     VAL_STRG(FORMAT := #CONVERT_FORMAT_TO_STRING,
              IN     := #date.MONTH,
              P      := #CONVERT_START_POSITION_MONTH,
              PREC   := #CONVERT_PRECISION,
              SIZE   := #CONVERT_SIZE_MONTH_DAY_HOUR_MINUTE_SECOND,
              OUT    => #tempString);     // DTL MONTH --> String --> #tempPosMonth

     VAL_STRG(FORMAT := #CONVERT_FORMAT_TO_STRING,
              IN     := #date.DAY,
              P      := #CONVERT_START_POSITION_DAY,
              PREC   := #CONVERT_PRECISION,
              SIZE   := #CONVERT_SIZE_MONTH_DAY_HOUR_MINUTE_SECOND,
              OUT    => #tempString);     // DTL DAY --> String --> #tempPosDay

     VAL_STRG(FORMAT := #CONVERT_FORMAT_TO_STRING,
              IN     := #date.HOUR,
              P      := #CONVERT_START_POSITION_HOUR,
              PREC   := #CONVERT_PRECISION,
              SIZE   := #CONVERT_SIZE_MONTH_DAY_HOUR_MINUTE_SECOND,
              OUT    => #tempString);     // DTL HOUR --> String --> #tempPosHour

     VAL_STRG(FORMAT := #CONVERT_FORMAT_TO_STRING,
              IN     := #date.MINUTE,
              P      := #CONVERT_START_POSITION_MINUTE,
              PREC   := #CONVERT_PRECISION,
              SIZE   := #CONVERT_SIZE_MONTH_DAY_HOUR_MINUTE_SECOND,
              OUT    => #tempString);     // DTL MINUTE --> String --> #tempPosMinute

     VAL_STRG(FORMAT := #CONVERT_FORMAT_TO_STRING,
              IN     := #date.SECOND,
              P      := #CONVERT_START_POSITION_SECOND,
              PREC   := #CONVERT_PRECISION,
              SIZE   := #CONVERT_SIZE_MONTH_DAY_HOUR_MINUTE_SECOND,
              OUT    => #tempString);     // DTL SECOND --> String --> #tempPosSecond

     VAL_STRG(FORMAT := #CONVERT_FORMAT_TO_STRING,
              IN     := #date.NANOSECOND,
              P      := #CONVERT_START_POSITION_NANOSECOND,
              PREC   := #CONVERT_PRECISION,
              SIZE   := #CONVERT_SIZE_NANOSECOND,
              OUT    => #tempString);     // DTL NANOSECOND --> String --> #tempPosNanosecond

     // Place separators at the right position in the string
     IF #separator = '' THEN
       #tempString[#SEPARATOR_POSITION_YEAR_MONTH] := #SEPARATOR_DATE;
       #tempString[#SEPARATOR_POSITION_MONTH_DAY] := #SEPARATOR_DATE;
     ELSE
       #tempString[#SEPARATOR_POSITION_YEAR_MONTH] := #separator;
       #tempString[#SEPARATOR_POSITION_MONTH_DAY] := #separator;
     END_IF;
     #tempString[#SEPARATOR_POSITION_HOUR_MINUTE] := #SEPARATOR_TIME;
     #tempString[#SEPARATOR_POSITION_MINUTE_SECOND] := #SEPARATOR_TIME;
     #tempString[#SEPARATOR_POSITION_SECOND_NANOSECOND] := #SEPARATOR_NANOSECOND;

     // Correcting the string, due to the conversion of a leading "0" value into a "blank".
     // Replacing of "blank" by "0"
     IF (#tempString[#CONVERT_START_POSITION_MONTH] = ' ') THEN
       #tempString[#CONVERT_START_POSITION_MONTH] := '0';
     END_IF;

     IF (#tempString[#CONVERT_START_POSITION_DAY] = ' ') THEN
       #tempString[#CONVERT_START_POSITION_DAY] := '0';
     END_IF;

     IF (#tempString[#CONVERT_START_POSITION_HOUR] = ' ') THEN
       #tempString[#CONVERT_START_POSITION_HOUR] := '0';
     END_IF;

     IF (#tempString[#CONVERT_START_POSITION_MINUTE] = ' ') THEN
       #tempString[#CONVERT_START_POSITION_MINUTE] := '0';
     END_IF;

     IF (#tempString[#CONVERT_START_POSITION_SECOND] = ' ') THEN
       #tempString[#CONVERT_START_POSITION_SECOND] := '0';
     END_IF;

     FOR #tempIndex := 0 TO #REPLACE_NANOSECOND_COUNT DO
       IF (#tempString[UINT_TO_SINT(#CONVERT_START_POSITION_NANOSECOND) + #tempIndex] = ' ') THEN
         #tempString[UINT_TO_SINT(#CONVERT_START_POSITION_NANOSECOND) + #tempIndex] := '0';
       ELSE
         EXIT;
       END_IF;
     END_FOR;
   END_REGION

   REGION OUTPUTS
     #LGF_DTLtoString_ISO := #tempString;
     // no error handling needed
     ENO := TRUE;
   END_REGION
END_FUNCTION